// TIA Portal project "etude cas final" (V16)

(* hardware
DEVICE "Station S71500/ET200MP_1"  S7-1500 station
   slot 0: "Châssis_0"  Rack  6ES7 590-1***0-0AA0
   slot 1: "PLC_1"  CPU 1511C-1 PN  6ES7 511-1CK01-0AB0  V2.8
      slot 3: "Ecran CPU_1"  6ES7591-1AA00-0AA0
      slot 32768: "Interface PROFINET_1"  X1
         slot 32769: "Port_1"  X1 P1
         slot 32770: "Port_2"  X1 P2
      slot 34817: "Virtual CP interface port_1"  Virtual CP interface port  Virtual CP interface port
DEVICE "HMI_1"  TP900 Comfort
   slot 0: "HMI_1"  TP900 Comfort  6AV2 124-0JC01-0AX0  16.0.0.0
   slot 1: "HMI_RT_1"  TP900 Comfort  6AV2 124-0JC01-0AX0  16.0.0.0
   slot 5: "HMI_1.IE_CP_1"  PROFINET Interface  16.0.0.0
      slot 1: "Interface PROFINET_1"  PROFINET Interface
         slot 1: "Port_1"  Port
         slot 2: "Port_2"  Port
   slot 7: "HMI_1.MPI/DP_CP_1"  MPI/DP Interface  16.0.0.0
*)

// ===== PLC "PLC_1"  CPU 1511C-1 PN =====

VAR_GLOBAL   // PLC tag table "Table de variables standard"
   "capteurb1" AT %IW0 : Int;
   "capteurb2" AT %IW2 : Int;
   "capteurb3" AT %IW4 : Int;
   "capteurb4" AT %IW6 : Int;
   "capteurp" AT %IW8 : Int;
   "stopv1" AT %I10.0 : Bool;
   "startv2" AT %I10.1 : Bool;
   "stopv2" AT %I10.2 : Bool;
   "startv3" AT %I10.3 : Bool;
   "stopv3" AT %I10.4 : Bool;
   "startv4" AT %I10.5 : Bool;
   "startv1" AT %I10.6 : Bool;
   "stopv4" AT %I10.7 : Bool;
   "vanne1" AT %Q4.0 : Bool;
   "vanne2" AT %Q4.1 : Bool;
   "vanne3" AT %Q4.2 : Bool;
   "vanne4" AT %Q4.3 : Bool;
   "Tag_1" AT %MD2 : Real;
   "Tag_2" AT %MD6 : Real;
   "Tag_3" AT %MD1 : Real;
   "Tag_4" AT %MD10 : Real;
   "Tag_5" AT %MD14 : Real;
   "Tag_6" AT %MD20 : Real;
   "Tag_7" AT %MD24 : Real;
   "Tag_8" AT %MD26 : Real;
   "Tag_9" AT %MD30 : Real;
   "Tag_10" AT %MD32 : Real;
   "Tag_11" AT %MD36 : Real;
   "pompe1" AT %Q4.4 : Bool;
   "pompe2" AT %Q4.5 : Bool;
END_VAR

ORGANIZATION_BLOCK "Main"   // OB1, LAD, ProgramCycle
TITLE = "Main Program Sweep (Cycle)"
{ S7_Optimized_Access := 'TRUE' }
VERSION : 0.1
   VAR_INPUT
      Initial_Call : Bool;   // Initial call of this OB
      Remanence : Bool;   // =True, if remanent data are available
   END_VAR
BEGIN

REGION Network 1
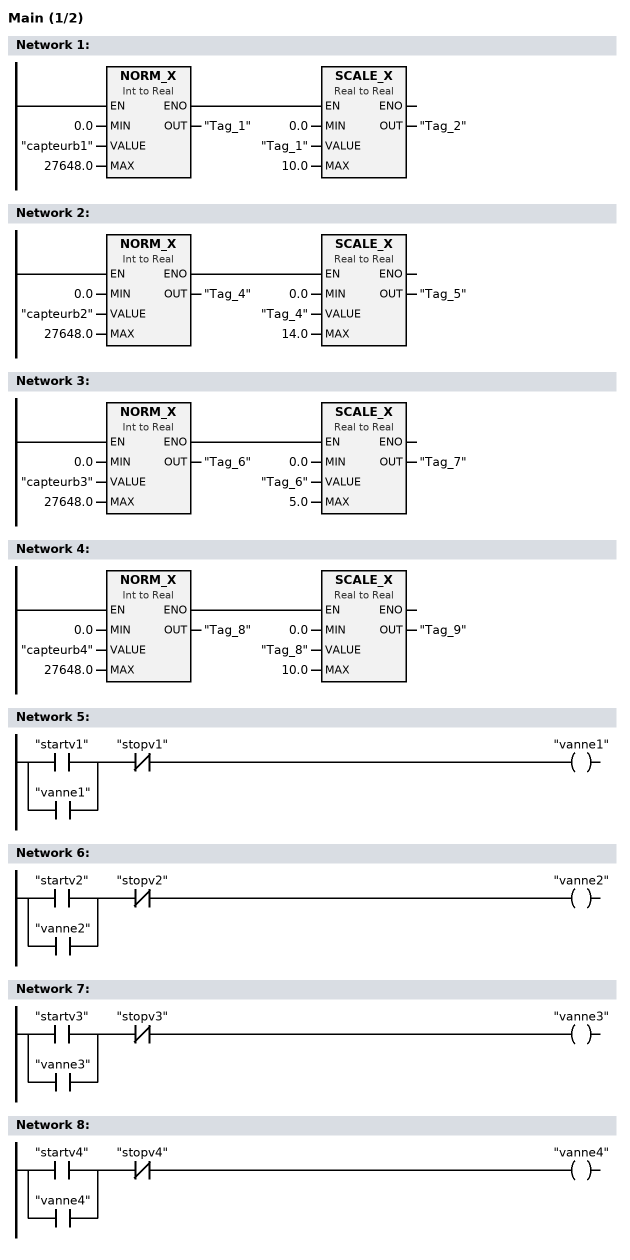
   RUNG wire#powerrail
      { S7_Templates := "[SrcType := Int, DestType := Real]" } Normalize(min := 0.0, value := "capteurb1", max := 27648.0, out => "Tag_1")
      { S7_Templates := "[SrcType := Real, DestType := Real]" } Scale(min := 0.0, value := "Tag_1", max := 10.0, out => "Tag_2")
   END_RUNG
   // the same network as SCL:
   "Tag_1" := NORM_X(MIN := 0.0, VALUE := "capteurb1", MAX := 27648.0);
   "Tag_2" := SCALE_X(MIN := 0.0, VALUE := "Tag_1", MAX := 10.0);
END_REGION

REGION Network 2
   RUNG wire#powerrail
      { S7_Templates := "[SrcType := Int, DestType := Real]" } Normalize(min := 0.0, value := "capteurb2", max := 27648.0, out => "Tag_4")
      { S7_Templates := "[SrcType := Real, DestType := Real]" } Scale(min := 0.0, value := "Tag_4", max := 14.0, out => "Tag_5")
   END_RUNG
   // the same network as SCL:
   "Tag_4" := NORM_X(MIN := 0.0, VALUE := "capteurb2", MAX := 27648.0);
   "Tag_5" := SCALE_X(MIN := 0.0, VALUE := "Tag_4", MAX := 14.0);
END_REGION

REGION Network 3
   RUNG wire#powerrail
      { S7_Templates := "[SrcType := Int, DestType := Real]" } Normalize(min := 0.0, value := "capteurb3", max := 27648.0, out => "Tag_6")
      { S7_Templates := "[SrcType := Real, DestType := Real]" } Scale(min := 0.0, value := "Tag_6", max := 5.0, out => "Tag_7")
   END_RUNG
   // the same network as SCL:
   "Tag_6" := NORM_X(MIN := 0.0, VALUE := "capteurb3", MAX := 27648.0);
   "Tag_7" := SCALE_X(MIN := 0.0, VALUE := "Tag_6", MAX := 5.0);
END_REGION

REGION Network 4
   RUNG wire#powerrail
      { S7_Templates := "[SrcType := Int, DestType := Real]" } Normalize(min := 0.0, value := "capteurb4", max := 27648.0, out => "Tag_8")
      { S7_Templates := "[SrcType := Real, DestType := Real]" } Scale(min := 0.0, value := "Tag_8", max := 10.0, out => "Tag_9")
   END_RUNG
   // the same network as SCL:
   "Tag_8" := NORM_X(MIN := 0.0, VALUE := "capteurb4", MAX := 27648.0);
   "Tag_9" := SCALE_X(MIN := 0.0, VALUE := "Tag_8", MAX := 10.0);
END_REGION

REGION Network 5
   RUNG wire#powerrail
      Contact( "startv1" )
      wire#w1
      I_Contact( "stopv1" )
      Coil( "vanne1" )
   END_RUNG
   RUNG wire#powerrail
      Contact( "vanne1" )
   END_RUNG wire#w1
   // the same network as SCL:
   "vanne1" := ("startv1" OR "vanne1") AND NOT "stopv1";
END_REGION

REGION Network 6
   RUNG wire#powerrail
      Contact( "startv2" )
      wire#w1
      I_Contact( "stopv2" )
      Coil( "vanne2" )
   END_RUNG
   RUNG wire#powerrail
      Contact( "vanne2" )
   END_RUNG wire#w1
   // the same network as SCL:
   "vanne2" := ("startv2" OR "vanne2") AND NOT "stopv2";
END_REGION

REGION Network 7
   RUNG wire#powerrail
      Contact( "startv3" )
      wire#w1
      I_Contact( "stopv3" )
      Coil( "vanne3" )
   END_RUNG
   RUNG wire#powerrail
      Contact( "vanne3" )
   END_RUNG wire#w1
   // the same network as SCL:
   "vanne3" := ("startv3" OR "vanne3") AND NOT "stopv3";
END_REGION

REGION Network 8
   RUNG wire#powerrail
      Contact( "startv4" )
      wire#w1
      I_Contact( "stopv4" )
      Coil( "vanne4" )
   END_RUNG
   RUNG wire#powerrail
      Contact( "vanne4" )
   END_RUNG wire#w1
   // the same network as SCL:
   "vanne4" := ("startv4" OR "vanne4") AND NOT "stopv4";
END_REGION

REGION Network 9
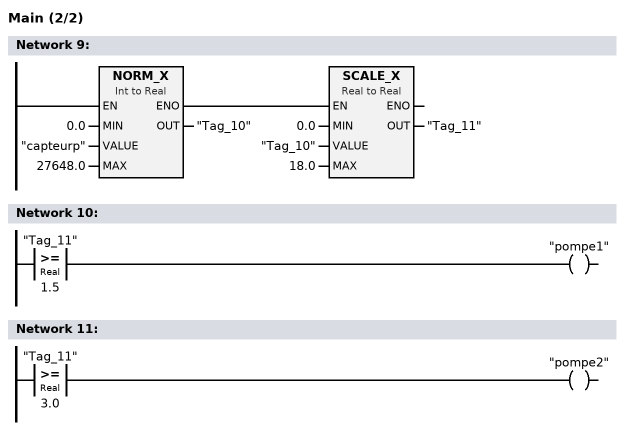
   RUNG wire#powerrail
      { S7_Templates := "[SrcType := Int, DestType := Real]" } Normalize(min := 0.0, value := "capteurp", max := 27648.0, out => "Tag_10")
      { S7_Templates := "[SrcType := Real, DestType := Real]" } Scale(min := 0.0, value := "Tag_10", max := 18.0, out => "Tag_11")
   END_RUNG
   // the same network as SCL:
   "Tag_10" := NORM_X(MIN := 0.0, VALUE := "capteurp", MAX := 27648.0);
   "Tag_11" := SCALE_X(MIN := 0.0, VALUE := "Tag_10", MAX := 18.0);
END_REGION

REGION Network 10
   RUNG wire#powerrail
      { S7_Templates := "SrcType := Real" } GE_Contact(in1 := "Tag_11", in2 := 1.5)
      Coil( "pompe1" )
   END_RUNG
   // the same network as SCL:
   "pompe1" := "Tag_11" >= 1.5;
END_REGION

REGION Network 11
   RUNG wire#powerrail
      { S7_Templates := "SrcType := Real" } GE_Contact(in1 := "Tag_11", in2 := 3.0)
      Coil( "pompe2" )
   END_RUNG
   // the same network as SCL:
   "pompe2" := "Tag_11" >= 3.0;
END_REGION
END_ORGANIZATION_BLOCK

(* ===== HMI "HMI_RT_1" =====
system functions are stored by id; their names below are inferred from use
connection "HMI_Liaison_1": ETHERNET, S7_1500_OMS

HMI tags "Table de variables standard"
   "Tag_2" : Real = PLC Tag_2 AT %MD6, 1 s
   "Tag_5" : Real = PLC Tag_5 AT %MD14, 1 s
   "Tag_7" : Real = PLC Tag_7 AT %MD24, 1 s
   "Tag_9" : Real = PLC Tag_9 AT %MD30, 1 s
   "Tag_11" : Real = PLC Tag_11 AT %MD36, 1 s
   "startv1" : Bool = PLC startv1 AT %I10.6, 1 s
   "stopv1" : Bool = PLC stopv1 AT %I10.0, 1 s
   "startv2" : Bool = PLC startv2 AT %I10.1, 1 s
   "stopv2" : Bool = PLC stopv2 AT %I10.2, 1 s
   "startv3" : Bool = PLC startv3 AT %I10.3, 1 s
   "stopv3" : Bool = PLC stopv3 AT %I10.4, 1 s
   "startv4" : Bool = PLC startv4 AT %I10.5, 1 s
   "stopv4" : Bool = PLC stopv4 AT %I10.7, 1 s
   "vanne1" : Bool = PLC vanne1 AT %Q4.0, 1 s
   "vanne2" : Bool = PLC vanne2 AT %Q4.1, 1 s
   "vanne3" : Bool = PLC vanne3 AT %Q4.2, 1 s
   "vanne4" : Bool = PLC vanne4 AT %Q4.3, 1 s
   "pompe1" : Bool = PLC pompe1 AT %Q4.4, 1 s
   "pompe2" : Bool = PLC pompe2 AT %Q4.5, 1 s

screen "Vue racine" 800x480, template "Modèle_1"
   Bar "Bargraphe_2" at 173,24 size 123x164; MinimumValue 0; MaximumValue 14
      ProcessValue <- "Tag_5"
   Bar "Bargraphe_3" at 516,20 size 74x103; MinimumValue 0
      ProcessValue <- "Tag_7"
   Bar "Bargraphe_4" at 690,20 size 89x126; MinimumValue 0; MaximumValue 10
      ProcessValue <- "Tag_9"
   Bar "Bargraphe_5" at 83,407 size 691x73; MinimumValue 0; MaximumValue 18
      ProcessValue <- "Tag_11"
   GraphicView "Vue de graphique_2" at 708,142 size 37x33; Picture "Graphique_4"
   GraphicView "Vue de graphique_7" at 556,139 size 23x22; Picture "Graphique_24"
   GraphicView "Vue de graphique_8" at 560,120 size 24x30; Picture "Graphique_4"
   GraphicView "Vue de graphique_10" at 83,129 size 15x21; Picture "Graphique_46"
   GraphicView "Vue de graphique_12" at 458,165 size 45x36; Picture "Graphique_49"
   GraphicView "Vue de graphique_13" at 469,147 size 43x28; Picture "Graphique_50"
   GraphicView "Vue de graphique_11" at 139,133 size 25x25; Picture "Graphique_51"
   GraphicView "Vue de graphique_15" at 139,145 size 31x111; Picture "Graphique_4"
   GraphicView "Vue de graphique_16" at 424,182 size 42x35; Picture "Graphique_52"
   GraphicView "Vue de graphique_9" at 146,248 size 33x32; Picture "Graphique_6"
   GraphicView "Vue de graphique_17" at 168,257 size 166x28; Picture "Graphique_46"
   GraphicView "Vue de graphique_18" at 321,248 size 38x32; Picture "Graphique_24"
   GraphicView "Vue de graphique_19" at 331,208 size 35x52; Picture "Graphique_4"
   GraphicView "Vue de graphique_20" at 339,182 size 37x33; Picture "Graphique_21"
   GraphicView "Vue de graphique_21" at 373,176 size 61x30; Picture "Graphique_25"
   GraphicView "Vue de graphique_22" at 413,207 size 44x37; Picture "Graphique_56"
   GraphicView "Vue de graphique_23" at 314,209 size 116x32; Picture "Graphique_46"
   GraphicView "Vue de graphique_24" at 231,201 size 33x33; Picture "Graphique_57"
   GraphicView "Vue de graphique_25" at 225,182 size 29x22; Picture "Graphique_4"
   GraphicView "Vue de graphique_27" at 426,233 size 38x180; Picture "Graphique_22"
   GraphicView "Vue de graphique_35" at 553,359 size 41x47; Picture "Graphique_76"
   GraphicView "Vue de graphique_36" at 572,214 size 40x44; Picture "Graphique_41"
   GraphicView "Vue de graphique_38" at 564,252 size 36x116; Picture "Graphique_4"
   GraphicView "Vue de graphique_39" at 604,205 size 195x39; Picture "Graphique_46"
   GraphicView "Vue de graphique_40" at 695,314 size 43x50; Picture "Graphique_41"
   GraphicView "Vue de graphique_41" at 721,304 size 79x44; Picture "Graphique_46"
   Button "Bouton_1" at 303,30 size 67x37; TextOff 'start v2'
      on Release: ResetBit("startv2")
      on Press: SetBit("startv2")
   Button "Bouton_2" at 303,70 size 68x37; TextOff 'stop v2'
      on Release: SetBit("stopv2")
      on Press: ResetBit("stopv2")
   Button "Bouton_3" at 87,25 size 67x37; TextOff 'start v1'
      on Release: ResetBit("startv1")
      on Press: SetBit("startv1")
   Button "Bouton_4" at 88,70 size 66x37; TextOff 'stop v1'
      on Release: SetBit("stopv1")
      on Press: ResetBit("stopv1")
   Button "Bouton_5" at 439,68 size 66x37; TextOff 'stop v3'
      on Release: SetBit("stopv3")
      on Press: ResetBit("stopv3")
   Button "Bouton_6" at 439,24 size 67x37; TextOff 'start v3'
      on Release: ResetBit("startv3")
      on Press: SetBit("startv3")
   Button "Bouton_7" at 613,27 size 67x37; TextOff 'start v4'
      on Release: ResetBit("startv4")
      on Press: SetBit("startv4")
   Button "Bouton_8" at 613,75 size 66x37; TextOff 'stop v4'
      on Release: SetBit("stopv4")
      on Press: ResetBit("stopv4")
   SymbolLibrary "Bibliothèque des icônes_1" at 485,284 size 70x124
      Appearance <- "pompe1"
   GraphicView "Vue de graphique_30" at 485,377 size 33x36; Picture "Graphique_75"
   GraphicView "Vue de graphique_37" at 487,409 size 28x67; Picture "Graphique_4"
   SymbolLibrary "Bibliothèque des icônes_2" at 608,283 size 70x124
      Appearance <- "pompe2"
   GraphicView "Vue de graphique_29" at 607,374 size 32x41; Picture "Graphique_75"
   GraphicView "Vue de graphique_31" at 608,409 size 28x61; Picture "Graphique_4"
   GraphicView "Vue de graphique_32" at 675,355 size 43x51; Picture "Graphique_76"
   SymbolLibrary "Bibliothèque des icônes_3" at 94,105 size 55x43
      Appearance <- "vanne1"
   SymbolLibrary "Bibliothèque des icônes_4" at 262,191 size 57x43
      Appearance <- "vanne2"
   SymbolLibrary "Bibliothèque des icônes_5" at 506,129 size 57x33
      Appearance <- "vanne3"
   SymbolLibrary "Bibliothèque des icônes_6" at 642,157 size 61x43
      Appearance <- "vanne4"
   GraphicView "Vue de graphique_3" at 696,169 size 42x31; Picture "Graphique_24"
   GraphicView "Vue de graphique_1" at 497,176 size 157x30; Picture "Graphique_46"
   TextField "Champ de texte_1" at 0,6 size 66x20; Text 'bassin 1'
   TextField "Champ de texte_2" at 204,0 size 66x20; Text 'bassin 2'
   TextField "Champ de texte_3" at 524,0 size 66x20; Text 'bassin 3'
   TextField "Champ de texte_4" at 708,1 size 66x20; Text 'bassin 4'
   TextField "Champ de texte_5" at 17,159 size 23x20; Text 'v1'
   TextField "Champ de texte_6" at 43,157 size 23x20; Text 'v2'
   TextField "Champ de texte_8" at 83,158 size 23x20; Text 'v3'
   TextField "Champ de texte_10" at 501,252 size 23x20; Text 'p1'
   TextField "Champ de texte_11" at 624,256 size 23x20; Text 'p2'
   Bar "Bargraphe_1" at 4,24 size 81x126; MinimumValue 0; MaximumValue 10
      ProcessValue <- "Tag_2"
   IOField "Champ d'E/S_1" at 29,25 size 33x24; FormatPattern 99
      ProcessValue <- "Tag_2"
   IOField "Champ d'E/S_2" at 221,26 size 33x23; FormatPattern 99
      ProcessValue <- "Tag_5"
   IOField "Champ d'E/S_3" at 542,20 size 22x22; FormatPattern 9
      ProcessValue <- "Tag_7"
   IOField "Champ d'E/S_4" at 718,22 size 30x23; FormatPattern 99
      ProcessValue <- "Tag_9"
   IOField "Champ d'E/S_5" at 111,409 size 23x25; FormatPattern 9
      ProcessValue <- "Tag_11"
   Ellipse "Ellipse_1" at 11,177 size 31x31
      Appearance <- "vanne1"
   Ellipse "Ellipse_2" at 44,178 size 31x31
      Appearance <- "vanne2"
   Ellipse "Ellipse_3" at 83,178 size 31x31
      Appearance <- "vanne3"
   Ellipse "Ellipse_4" at 9,225 size 31x31
      Appearance <- "vanne4"
   TextField "Champ de texte_7" at 12,206 size 23x20; Text 'v4'
   Ellipse "Ellipse_5" at 43,225 size 32x31
      Appearance <- "pompe1"
   Ellipse "Ellipse_6" at 83,226 size 32x31
      Appearance <- "pompe2"
   TextField "Champ de texte_9" at 48,207 size 23x20; Text 'p1'
   TextField "Champ de texte_12" at 90,206 size 23x20; Text 'p2'
   SymbolLibrary "Bibliothèque des icônes_7" at 117,159 size 9x114
   SymbolLibrary "Bibliothèque des icônes_8" at 0,266 size 126x8
   SymbolLibrary "Bibliothèque des icônes_9" at 0,154 size 126x8
   SymbolLibrary "Bibliothèque des icônes_10" at 0,161 size 9x114
*)